FUNCTION_BLOCK PUBLIC fbSealingCorkAssKeyencePN EXTENDS fbStFixBaseTemplate IMPLEMENTS I_Fixture 

VAR
	fbVisionSensor: fbKeyenceIVProfinetCtrl;
	I_Vision: I_VisionSensorSTD;
	iTriggerRepeats: INT;
	bErrorBVS: BOOL;
	bOring 	: BOOL;
	bCap		: BOOL;
	bOringWidth : BOOL;
	iDetecitonPick	: INT;
END_VAR
VAR PERSISTENT
	stParams	:	 stKeyenceInspectionParams;
END_VAR

fbVisionSensor(iInspectionToActive:=stParams.iProgramNumber);
I_Vision := fbVisionSensor;
stParams.bInspectionEnable S=  GVL.fbUserLogin.nUserRole <> nSQL_UserRoles.Maintenance;
CASE iWorkStep OF
	0:		// Powrót do stanu początkowego (ustawienie zmiennych)
		bResetMethod := bQReady := bQBusy := bQError := FALSE;
		fbVisionSensor.bTrigger := FALSE;
		IF NOT bLock AND NOT bRelease THEN
			fbTON(IN:= FALSE);
			iWorkStep := 1;
		END_IF
			
	1: 		// Sprawdzenie czy siłowniki są w dobrej pozycji itp.
		fbTON(IN:= TRUE, PT:= T#2S);
		bQLocked := FALSE;
		iWorkStep := 5;
	
	5:		// Oczekiwanie na nowy rozkaz
		bResetMethod:= bReleaseMethod:= bAuxOperMethod:= bLockMethod := FALSE;
		bQReady := TRUE;
		actCheckForNewOrder();
		
	10:		// Blokowanie kowadła
		bQError := FALSE;
		IF stParams.bInspectionEnable THEN
			nQErrorId := iTriggerRepeats := 0;
			iWorkStep := 12;
		ELSE
			iWorkStep := 16;
		END_IF
		
	12:		// Oczekiwanie na zakończenie detekcji
		IF I_Vision.mNewInspection(bError => bErrorBVS, bOut1=> bOring, bOut2=> bCap, bOut3 => bOringWidth) THEN
			iDetecitonPick.0 := NOT bOring;			//0-1
			iDetecitonPick.1 := NOT bCap;			//0-2
			iDetecitonPick.2 := NOT bOringWidth;	//0-4
			IF NOT bErrorBVS THEN		// Balluff odpowiedział
				IF bOring AND bCap AND bOringWidth THEN		// Wszystko wykryte
					iWorkStep := 16;
				ELSE		// NIe wyszystko wykryte
					IF iTriggerRepeats >= stParams.iMaxTrigRepeats THEN		// Wykonano powtórne zdjęcie
						CASE iDetecitonPick OF
							0:
								mNewError(nSealingCorkAssKeyencePN_ErrorCodes.BadSealingCorkAssembly);
							1:
								mNewError(nSealingCorkAssKeyencePN_ErrorCodes.LackOfOring);
							2:
								mNewError(nSealingCorkAssKeyencePN_ErrorCodes.CapNotDetected);
							3:
								mNewError(nSealingCorkAssKeyencePN_ErrorCodes.CapNotDetectedAndNoOring);
							4:
								mNewError(nSealingCorkAssKeyencePN_ErrorCodes.WrongOringWidth);
							5:
								mNewError(nSealingCorkAssKeyencePN_ErrorCodes.LackOfOring);
							6:
								mNewError(nSealingCorkAssKeyencePN_ErrorCodes.WrongOringWidthAndCapNotDetected);
							7:
								mNewError(nSealingCorkAssKeyencePN_ErrorCodes.BadSealingCorkAssembly);
						END_CASE
					ELSE		// Wykonaj powtórne zdjęcie
						iTriggerRepeats := iTriggerRepeats + 1;
						fbTON(IN:= FALSE);
						iWorkStep := 14;
					END_IF
				END_IF
			ELSE		// brak odpowiedzi Balluffa
				mNewError(nSealingCorkAssKeyencePN_ErrorCodes.SensorNotReady);
			END_IF
		END_IF
	14:		// Oczekiwanie oraz powtórna próba znalezienia
		fbTON(IN:= TRUE, PT:= T#200MS);
		IF fbTON.Q THEN
			fbTON(IN:= FALSE);
			iWorkStep := 12;
		END_IF
	16:		// Wszystko wykryte OK
		bQError := bQBusy := FALSE;
		iWorkStep := 5;
		
	20:		// Dodatkowa operacja
		bQBusy := FALSE;
		bQLocked := FALSE;		
		iWorkStep := 5;
	
	30:		// Zwalnianie kowadła
		bQBusy := FALSE;
		bQLocked := FALSE;		
		iWorkStep := 5;
	
	50:		// Manual work coordination
		fbTON(IN:= TRUE, PT:= T#15M);
		IF NOT bManualWork OR fbTON.Q THEN
			fbTON(IN:= FALSE);
			bManualWork := FALSE;
			iWorkStep := 0;
		END_IF	
		
	90:		// Błąd w pracy kowadła
		bQBusy := bQReady:= bQAlarm := FALSE;
		bQError := TRUE;
		fbVisionSensor.bTrigger := fbVisionSensor.bReadActualInspection := fbVisionSensor.bChangeInspection := FALSE;
		iWorkStep := 95;
		
	91:
		bQBusy := bQReady := FALSE;
		bQAlarm := TRUE;
		fbVisionSensor.bTrigger := fbVisionSensor.bReadActualInspection := fbVisionSensor.bChangeInspection := FALSE;
		iWorkStep := 95;

	
	95:
		IF bRelease OR bResetMethod THEN
			bQError := FALSE;
			nQErrorId := iWorkStep := 0;
		END_IF

	ELSE
		mNewError(nSealingCorkAssKeyencePN_ErrorCodes.ProgramConfigError);			
END_CASE

stParams.bInspectionEnable := TRUE;

END_FUNCTION_BLOCK

(* stored: Version 1.1.0.1, ProductVersion 3.1.4024.15
   POU fbSealingCorkAssKeyencePN: Id {a2e71178-4ee5-46d0-be3f-d542ea62a160}, SpecialFunc None *)
